// TIA Portal V16 export
// export: Created 2022-11-01T21:54:09.2027362Z, ExportSetting WithDefaults, DisplayName Totally Integrated Automation Portal, DisplayVersion V16, DisplayName TIA Portal Version Control Interface, DisplayVersion V16, DisplayName TIA Portal Openness, DisplayVersion V16, DisplayName SINAMICS Startdrive Advanced, DisplayVersion V16, DisplayName SINAMICS Startdrive G130, G150, S120, S150, SINAMICS MV, S210, DisplayVersion V16, DisplayName SINAMICS Startdrive G110M, G120, G120C, G120D, G120P, DisplayVersion V16, DisplayName STEP 7 Professional, DisplayVersion V16, DisplayName STEP 7 Safety, DisplayVersion V16, DisplayName WinCC Professional, DisplayVersion V16
VAR_GLOBAL   // PLC tag table "AO C600"
   qTV617 AT %QW210 : Int;
   qTV632 AT %QW212 : Int;
   "qTV640-1" AT %QW214 : Int;
   "qTV640-2" AT %QW216 : Int;
   "qTV642-1" AT %QW218 : Int;
   "qTV642-2" AT %QW220 : Int;
   "qPV602-1" AT %QW190 : Int;
   "qPV602-2" AT %QW192 : Int;
   qPV603 AT %QW194 : Int;
   qPV604 AT %QW196 : Int;
   "qPV609-1" AT %QW198 : Int;
   "qPV609-2" AT %QW200 : Int;
   qPV612 AT %QW202 : Int;
   qPV618 AT %QW204 : Int;
   qPV619 AT %QW206 : Int;
   qLV604 AT %QW182 : Int;
   qLV611 AT %QW184 : Int;
   qLV615 AT %QW186 : Int;
   qLV617 AT %QW188 : Int;
   qFV604 AT %QW138 : Int;
   qFV612 AT %QW140 : Int;
   qFV615 AT %QW142 : Int;
   qFV618 AT %QW144 : Int;
   qFV619 AT %QW146 : Int;
   qFV620 AT %QW148 : Int;
   "qUTV640-1" AT %QW224 : Int;
   "qUTV640-2" AT %QW226 : Int;
   "qUTV642-1" AT %QW228 : Int;
   "qUTV642-2" AT %QW230 : Int;
   qUFV612 AT %QW222 : Int;
   qH5_H6 AT %QW152 : Int;
   qH13 AT %QW150 : Int;
   "qH61/1_H61/2" AT %QW178 : Int;
   "qH62/1_H62/2" AT %QW180 : Int;
   "qH601/1" AT %QW154 : Int;
   "qH601/2" AT %QW156 : Int;
   "qH601/3" AT %QW158 : Int;
   "qH601/4" AT %QW160 : Int;
   "qH601/5" AT %QW162 : Int;
   "qH601/6" AT %QW164 : Int;
   "qH601/7" AT %QW166 : Int;
   "qH602/1" AT %QW168 : Int;
   "qH602/2" AT %QW170 : Int;
   "qH602/3" AT %QW172 : Int;
   "qH602/4" AT %QW174 : Int;
   "qH602/5" AT %QW176 : Int;
   qPV621 AT %QW208 : Int;
   "qBX601/1-1" AT %QW100 : Int;
   "qBX601/1-3" AT %QW102 : Int;
   "qBX601/1-5" AT %QW104 : Int;
   "qBX601/2-1" AT %QW106 : Int;
   "qBX601/2-3" AT %QW108 : Int;
   "qBX601/2-5" AT %QW110 : Int;
   "qBX602/1-1" AT %QW112 : Int;
   "qBX602/1-3" AT %QW114 : Int;
   "qBX602/1-5" AT %QW116 : Int;
   "qBX602/2-1" AT %QW118 : Int;
   "qBX602/2-3" AT %QW120 : Int;
   "qBX602/2-5" AT %QW122 : Int;
   "qBX602/3-1" AT %QW124 : Int;
   "qBX602/3-3" AT %QW126 : Int;
   "qBX602/3-5" AT %QW128 : Int;
   "qBX603/1-1" AT %QW130 : Int;
   "qBX603/1-3" AT %QW132 : Int;
   "qBX603/2-1" AT %QW134 : Int;
   "qBX603/2-3" AT %QW136 : Int;
END_VAR
